TYPE ST_LogLevelHeaders :
STRUCT
	Error	: STRING := '<Error> ';
	Warning	: STRING := '<Warning> ';
	Info	: STRING := '<Info> ';
END_STRUCT
END_TYPE

(* stored: Version 1.1.0.1, ProductVersion 3.1.4024.13
   DUT ST_LogLevelHeaders: Id {15a20e3d-fccd-0b61-1820-6f316ce0fdbd} *)
